(* PLC project CoDeSys External Library Template, WAGO e!COCKPIT e!COCKPIT, author 3S - Smart Software Solutions GmbH *)
(* stored: creationDateTime 2019-10-29T12:22:40.4663149, version 3.5.5.30, modificationDateTime 2019-10-24T14:40:07.960949, organization 3S - Smart Software Solutions GmbH *)
(* Library project template with all possible element types, docu and a sample project structure *)

(* values of enumPPPSSilownikTrybPracy: Manualny: Tryb pracy ręcznej; Automatyczny: Tryb pracy automatycznej *)

(* Autor: Artur Wyszomirski, 2018-09-25-AW Prawa majątkowe: Solwena Sp. z o.o., Aktualizacje: Opis: enum służy do obsługi Trybów pracy fb siłownika SABp (HRU0) na budynkach PPP Sopot (ENGIE) *)
{attribute 'qualified_only'}
{attribute 'strict'}
TYPE enumPPPSSilownikTrybPracy : (Manualny := 0, Automatyczny := 1);
END_TYPE
